FUNCTION_BLOCK FB_Lamp
VAR_INPUT
END_VAR
VAR_OUTPUT
END_VAR
VAR
	Key				AT %I* 	: BOOL;
	Lamp			AT %Q* 	: BOOL;
	rtKey: R_TRIG;
END_VAR


	rtKey(CLK:= Key, Q=> );
	IF rtKey.Q THEN
		Lamp		:=	NOT Lamp;
	END_IF

END_FUNCTION_BLOCK

(* stored: Version 1.1.0.1, ProductVersion 3.1.4024.12
   POU FB_Lamp: Id {5abcbe38-7ba1-4731-834c-dc3acbe917e9}, SpecialFunc None *)
